// TwinCAT 3 PLC project PLC
// ProgramVersion: 3.1.4026.20
// libraries:
//   Tc2_Standard, * (Beckhoff Automation GmbH)
//   Tc2_System, * (Beckhoff Automation GmbH)
// project tree:
//   DUTs/ ST_HmiRow.TcDUT
//   GVLs/ HMI.TcGVL
//   / PlcTask.TcTTO
//   POUs/ MAIN.TcPOU
// real-time tasks:
//   TASK PlcTask: cycle T#10ms, priority 20, ADS port 350

CONFIGURATION PLC
    RESOURCE PLC ON TwinCAT3
        TASK PlcTask(INTERVAL := T#10ms, PRIORITY := 20);
        PROGRAM MAIN WITH PlcTask : MAIN;
    END_RESOURCE
END_CONFIGURATION

// ---- DUTs/ST_HmiRow.TcDUT
TYPE ST_HmiRow :
STRUCT
    nIndex : UINT;
    sName : STRING(40);
    lrValue : LREAL;
    bEnabled : BOOL;
    sUnit : STRING(16);
    sSource : STRING(16);
END_STRUCT
END_TYPE

// ---- GVLs/HMI.TcGVL
{attribute 'qualified_only'}
VAR_GLOBAL
    aRows : ARRAY[1..8] OF ST_HmiRow := [
        (nIndex := 1, sName := 'SpeedSetpoint', lrValue := 120.0, bEnabled := TRUE, sUnit := 'mm/s', sSource := 'PLC'),
        (nIndex := 2, sName := 'PressureLimit', lrValue := 5.5, bEnabled := TRUE, sUnit := 'bar', sSource := 'PLC'),
        (nIndex := 3, sName := 'BatchCount', lrValue := 12.0, bEnabled := TRUE, sUnit := 'pcs', sSource := 'PLC'),
        (nIndex := 4, sName := 'Temperature', lrValue := 36.5, bEnabled := FALSE, sUnit := 'degC', sSource := 'PLC'),
        (nIndex := 5, sName := 'VacuumLevel', lrValue := -0.65, bEnabled := TRUE, sUnit := 'bar', sSource := 'PLC'),
        (nIndex := 6, sName := 'CycleDelay', lrValue := 250.0, bEnabled := FALSE, sUnit := 'ms', sSource := 'PLC'),
        (nIndex := 7, sName := 'RetryLimit', lrValue := 3.0, bEnabled := TRUE, sUnit := 'count', sSource := 'PLC'),
        (nIndex := 8, sName := 'RecipeNumber', lrValue := 1.0, bEnabled := TRUE, sUnit := 'id', sSource := 'PLC')
    ];
    nActiveRowCount : UINT := 8;
    nLastChangedIndex : UINT := 0;
    bCommitRequested : BOOL := FALSE;
END_VAR

// ---- POUs/MAIN.TcPOU
PROGRAM MAIN
VAR
    nIndex : UINT;
END_VAR

IF HMI.bCommitRequested THEN
    FOR nIndex := 1 TO HMI.nActiveRowCount DO
        HMI.aRows[nIndex].nIndex := nIndex;
        HMI.aRows[nIndex].sSource := 'PLC';
    END_FOR

    HMI.nLastChangedIndex := HMI.nActiveRowCount;
    HMI.bCommitRequested := FALSE;
END_IF

END_PROGRAM
